// TIA Portal V17 export
// export: Created 2026-10-01T22:11:08.0288669Z, ExportSetting WithDefaults, DisplayName Totally Integrated Automation Portal, DisplayVersion V17, DisplayName TIA Portal Openness, DisplayVersion V17, DisplayName TIA Portal Version Control Interface, DisplayVersion V17, DisplayName SINAMICS Startdrive Advanced, DisplayVersion V17, DisplayName SINAMICS Startdrive G130, G150, S120, S150, SINAMICS MV, G220, S200, S210, DisplayVersion V17, DisplayName SINAMICS Startdrive G110M, G120, G120C, G120D, G120P, G115D, DisplayVersion V17, DisplayName STEP 7 Professional, DisplayVersion V17, DisplayName STEP 7 Safety, DisplayVersion V17, DisplayName WinCC Basic/Comfort/Advanced, DisplayVersion V17, DisplayName WinCC Unified, DisplayVersion V17
FUNCTION_BLOCK "ZZ_LadTest_Cnt"   // FB31, LAD
{ S7_Optimized_Access := 'TRUE' }
VERSION : 0.1
// stored: AutoNumber true, IsIECCheckEnabled false, IsRetainMemResEnabled false, MemoryReserve 100, SetENOAutomatically false, UDAEnableTagReadback false
   VAR_INPUT
      Pulse : Bool;
      Rst : Bool;
   END_VAR
   VAR_OUTPUT
      Hit : Bool;
      Zero : Bool;
   END_VAR
   VAR RETAIN
      Up : CTU_INT;
      Dn : CTD_INT;
   END_VAR
BEGIN

REGION Network 1
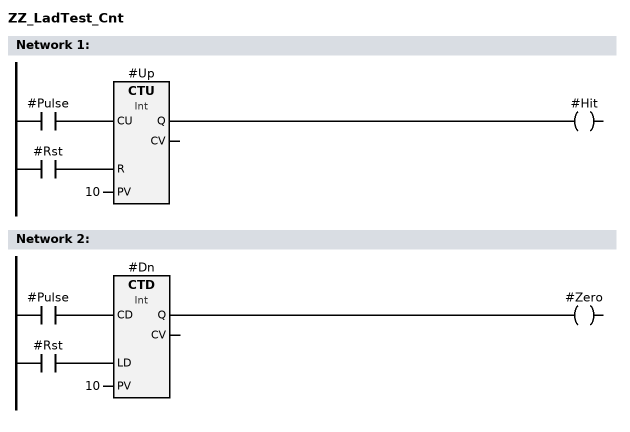
   RUNG wire#powerrail
      Contact( #Pulse )
      { S7_Templates := "value_type := Int" } #Up.CTU(r := wire#w1, pv := 10, cv =>)
      Coil( #Hit )
   END_RUNG
   RUNG wire#powerrail
      Contact( #Rst )
   END_RUNG wire#w1
   // the same network as SCL:
   #Up(CU := #Pulse, R := #Rst, PV := 10);   // CTU
   #Hit := #Up.Q;
END_REGION

REGION Network 2
   RUNG wire#powerrail
      Contact( #Pulse )
      { S7_Templates := "value_type := Int" } #Dn.CTD(ld := wire#w1, pv := 10, cv =>)
      Coil( #Zero )
   END_RUNG
   RUNG wire#powerrail
      Contact( #Rst )
   END_RUNG wire#w1
   // the same network as SCL:
   #Dn(CD := #Pulse, LD := #Rst, PV := 10);   // CTD
   #Zero := #Dn.Q;
END_REGION
END_FUNCTION_BLOCK
